# EPICS substitutions: ek9000App/Db/EL3122.substitutions
file EL3122.template
{       pattern
        {
                TERMINAL,

        }
        {
        }
}
